(* PLC project Mx9_v_0_3_3.project, CODESYS CODESYS V3.5 SP5 Patch 5 *)
(* stored: creationDateTime 2017-10-23T23:21:49.9734832, modificationDateTime 2017-10-21T13:03:26.8127651 *)

TYPE component : STRUCT
  step : STRING;
  code : STRING;
  name : STRING;
  weight : STRING;
  roughWeight : STRING;
END_STRUCT;
END_TYPE

PROGRAM PLC_PRG
  VAR
    bStatInit : BOOL;
    bStatStandby : BOOL;
    bStatSettings : BOOL;
    bStatPause : BOOL;
    bStatLoad : BOOL;
    bLog : BOOL;
    bManualMode : BOOL;
    rTara : REAL;
    bTara : BOOL;
    rClean : REAL;
    precisionTimer : Standard.TON;
    sConsole : STRING := 'Console output';
    dfa : dfa;  (* classes *)
    switch : switch;
    list : list;
    logger : logger;
    recMan : RecipeManCommands;
    filter : filter;
  END_VAR

                    //a_read();
//b_tara();
rClean := filter.clean( rWeight );
blinkJob();
// test visu pumps to pump tubes link effect
FOR i := 1 TO 4 DO
	IF pumps[i] AND switch.isPumpRun() THEN pump_tubes[i] := TRUE; END_IF
END_FOR

CASE dfa.iStatementCode OF //набор состояний системы	
	0:// INIT
			blink ( TIMEHIGH := T#1S, TIMELOW := T#1S );
			bStatInit := TRUE;
			logger.init();
			recMan.WriteRecipe( namesGroup, namesFile );
			recMan.WriteRecipe( 'settings', filter_settngs_filename );
			dfa.exec('checked');
			
		IF dfa.bQuitStat THEN // EXIT
			bStatInit := FALSE;
		END_IF
		
	1:// STANDBY
		IF dfa.bEnterStat THEN
			 // ======== ENTER =========== //
			  //StatStandby := TRUE;
			//logger.writeStat( 'Enter standby mode');
			//IF logger.done THEN
				dfa.endEnter();
			//END_IF
			// ======== END ENTER ======== //
		END_IF
		
		//---------- BODY -----------//
		
		//------- END_BODY ----------//
		
		IF dfa.bQuitStat THEN 
		// ========== EXIT =========== //
			;
		// ======== END EXIT ======== //
		END_IF
		
	2:// SETTINGS
		IF dfa.bEnterStat THEN
			 // ======== ENTER =========== //
			 
			 
			dfa.endEnter();
			// ======== END ENTER ======== //
		END_IF
		
		//---------- BODY -----------//
		
		//------- END_BODY ----------//
		
		IF dfa.bQuitStat THEN 
		// ========== EXIT =========== //
		
		
		// ======== END EXIT ======== //
		END_IF

	3:// PROGRAMMING
		IF dfa.bEnterStat THEN
			 // ======== ENTER =========== //
			 
			 
			dfa.endEnter();
			// ======== END ENTER ======== //
		END_IF
		
		//---------- BODY -----------//
		
		//------- END_BODY ----------//
		
		IF dfa.bQuitStat THEN 
		// ========== EXIT =========== //
		
		
		// ======== END EXIT ======== //
		END_IF
		
	4:// CHOOSING
		IF dfa.bEnterStat THEN
			 // ======== ENTER =========== //
			dfa.endEnter();
			// ======== END ENTER ======== //
		END_IF
		
		//---------- BODY -----------//
		list.man_cmp_mode_job();
		//------- END_BODY ----------//
		
		IF dfa.bQuitStat THEN 
		// ========== EXIT =========== //
			IF bManualMode THEN
				list.man_counters_init();
			END_IF		
		// ======== END EXIT ======== //
		END_IF

	5:// ROUGH_LOADING
		IF dfa.bEnterStat THEN
			 // ======== ENTER =========== //
			IF bManualMode THEN 
				IF manWeightLimit = 0 THEN					
						dfa.exec('back'); 
					ELSE
						switch.on( componentNames[ i_man_count ], TRUE );
				END_IF
				
			END_IF
			 
			dfa.endEnter();
			// ======== END ENTER ======== //
		END_IF
		
		//---------- BODY -----------//
		IF bPause THEN dfa.exec('pause'); END_IF
		
		IF bManualMode THEN
			rWeight := rWeight + 0.01;
			list.man_mode_count();
			IF rWeight - rWeight_c_p >= ( manWeightLimit - manWeightPrecise ) THEN
				dfa.exec( 'done' );
			END_IF
		END_IF
		//------- END_BODY ----------//
		
		IF dfa.bQuitStat THEN 
		// ========== EXIT =========== //
		switch.allOff();
		
		// ======== END EXIT ======== //
		END_IF

	6:// PRECISE_LOADING
		IF dfa.bEnterStat THEN
			 // ======== ENTER =========== //
			dfa.endEnter();
			// ======== END ENTER ======== //
		END_IF
		
		//---------- BODY -----------//
		IF bPause THEN dfa.exec('pause'); END_IF
		
		IF bManualMode THEN
			precisionTimer( IN := TRUE, PT := T#5S );
			IF precisionTimer.Q THEN
				switch.on( componentNames[ i_man_count ], FALSE );
				rWeight := rWeight + 0.005;
				list.man_mode_count();
			END_IF
			IF rWeight - rWeight_c_p >= ( manWeightLimit ) THEN
				dfa.exec( 'listEnd' );
			END_IF
		END_IF
		//------- END_BODY ----------//
		
		IF dfa.bQuitStat THEN 
		// ========== EXIT =========== //
		precisionTimer( IN := FALSE );
		switch.allOff();
		
		// ======== END EXIT ======== //
		END_IF

	7:// DONE
		IF dfa.bEnterStat THEN
			 // ======== ENTER =========== //
			 
			dfa.endEnter();
			// ======== END ENTER ======== //
		END_IF		
		//---------- BODY -----------//
		
		//------- END_BODY ----------//
		
		IF dfa.bQuitStat THEN 
		// ========== EXIT =========== //
		
		
		// ======== END EXIT ======== //
		END_IF

	8:// PAUSE
		IF dfa.bEnterStat THEN
			 // ======== ENTER =========== //
				switch.allOff();
			 	logger.writeStat('Pause mode activated');
			 IF logger.done THEN
				dfa.endEnter();
			 END_IF
			// ======== END ENTER ======== //
		END_IF
		
		//---------- BODY -----------//
		IF NOT bPause THEN
			dfa.exec('back');			
			//switch.on( switch.sLastCode, switch.bLastRough );
		END_IF
		
		//------- END_BODY ----------//
		
		IF dfa.bQuitStat THEN 
		// ========== EXIT =========== //
		
		
		// ======== END EXIT ======== //
		END_IF

	ELSE	// состояние по-умолчанию
		
END_CASE
IF dfa.bQuitStat THEN // EXIT STATEMENT
	stats[dfa.iStatementCode] := FALSE;
	dfa.finishTransition();
	stats[dfa.iStatementCode] := TRUE;
END_IF
y_mach_table();
z_write();
                  

ACTION blinkJob:
                        IF switch.isPumpRun() THEN 
	blink( ENABLE := TRUE );		
	pumps[ switch.idxPump ] := blink.OUT ;
ELSE
	blink( ENABLE := FALSE );
END_IF
                      
END_ACTION

ACTION a_read:
                        rWeight := MV110_1TD.RdfF1 - rTara;
                      
END_ACTION

ACTION z_write:
                        iOutDiscrets := switch.iOut;
                      
END_ACTION

ACTION y_mach_table:
                        IF bManualMode THEN
	switch.matchTable();
END_IF;
                      
END_ACTION

ACTION b_tara:
                        IF bTara THEN
	rTara := MV110_1TD.RdfF1;
	bTara := FALSE;
END_IF
                      
END_ACTION
END_PROGRAM

FUNCTION_BLOCK dfa
  VAR_OUTPUT
    iStatementCode : INT;
    bEnterStat : BOOL;
    bQuitStat : BOOL;
  END_VAR
  VAR
    sCrntStatement : STRING := 'INIT';
    sPrevStatement : STRING;
    i : INT := 0;
    iFROM : INT := 0;
    iTRANSITION : INT := 1;
    iTO : INT := 2;
    arStatements : ARRAY[0..99] OF STRING := ['INIT', 'STANDBY', 'SETTINGS', 'PROGRAMMING', 'CHOOSING', 'ROUGH_LOADING', 'PRECISE_LOADING', 'DONE', 'PAUSE'];
    arTransitionTable : ARRAY[0..99, 0..2] OF STRING := ['INIT', 'checked', 'STANDBY', 'STANDBY', 'set', 'SETTINGS', 'STANDBY', 'start', 'CHOOSING', 'STANDBY', 'pause', 'PAUSE', 'SETTINGS', 'program', 'PROGRAMMING', 'SETTINGS', 'exit', 'STANDBY', 'PROGRAMMING', 'exit', 'STANDBY', 'PROGRAMMING', 'init', 'INIT', 'CHOOSING', 'exit', 'STANDBY', 'CHOOSING', 'load', 'ROUGH_LOADING', 'ROUGH_LOADING', 'pause', 'PAUSE', 'ROUGH_LOADING', 'done', 'PRECISE_LOADING', 'ROUGH_LOADING', 'listEnd', 'DONE', 'PRECISE_LOADING', 'next', 'ROUGH_LOADING', 'PRECISE_LOADING', 'pause', 'PAUSE', 'PRECISE_LOADING', 'listEnd', 'DONE', 'DONE', 'again', 'CHOOSING', 'DONE', 'exit', 'STANDBY', 'PAUSE', 'back', ''];
  END_VAR

                    
                  

{attribute 'object_name' := 'endEnter'}
METHOD endEnter
                          bEnterStat := FALSE;
                        
END_METHOD

{attribute 'object_name' := 'exec'}
METHOD exec
  VAR_INPUT
    sTransition : STRING;
  END_VAR
                          FOR i:= 0 TO 99 DO
	IF arTransitionTable[i, iFROM] = '' THEN
		RETURN;
	END_IF
	IF arTransitionTable[i, iFROM] = sCrntStatement AND arTransitionTable[i, iTRANSITION] = sTransition THEN
		
		sCrntStatement := SEL ( sTransition = 'back', arTransitionTable[i, iTO], sPrevStatement );
		
		sPrevStatement := arTransitionTable[i, iFROM];
		bQuitStat := TRUE;
		RETURN;
	END_IF
END_FOR
                        
END_METHOD

{attribute 'object_name' := 'finishTransition'}
METHOD finishTransition
                          FOR i:= 0 TO 99 DO
	IF arStatements[i] = '' THEN
		RETURN;		
	END_IF
	IF arStatements[i] = sCrntStatement THEN
		iStatementCode := i;
		bQuitStat := FALSE;
		bEnterStat := TRUE;
		RETURN;
	END_IF
END_FOR
                        
END_METHOD
END_FUNCTION_BLOCK

(* Набор переключателей *)
FUNCTION_BLOCK switch
  VAR_INPUT
    iIn : INT;
  END_VAR
  VAR_OUTPUT
    iOut : INT;
    idxPump : INT;
    sLastCode : STRING;
    bLastRough : BOOL;
  END_VAR
  VAR
    i : INT;
  END_VAR

                    
                  

(* выключает все 16 переключателей *)
{attribute 'object_name' := 'allOff'}
METHOD allOff
                          iOut := 0;
FOR i := 1 TO 11 DO
	IF i < 5 THEN
		pumps[ i ] := FALSE;
		pump_tubes[ i ] := FALSE;
	END_IF
	IF i < 10 THEN
		component_boxes[ i ] := FALSE;
	END_IF
	valves[ i ] := FALSE;
END_FOR
bPrecise := FALSE;
bRough := FALSE;
idxPump := 0;
                        
END_METHOD

(* устанавливает выключатели в ON *)
{attribute 'object_name' := 'on'}
METHOD on
  VAR_INPUT
    code : STRING;
    rough : BOOL;
  END_VAR
                          bRough := rough;
bPrecise := NOT rough;

sLastCode := code;
bLastRough := rough;

CASE getCodeIdx( code ) OF //набор переключателей в зависимости от кода
	1:	
			component_boxes[1] := TRUE;
			valves[1]	:= TRUE;
			valves[8]	:= TRUE;
			pump_tubes[1] := TRUE;
			idxPump := 1;			
	2:
			component_boxes[2] := TRUE;
			valves[2]	:= TRUE;
			valves[8]	:= TRUE;
			pump_tubes[1] := TRUE;
			idxPump := 1;			
	3:
			component_boxes[3] := TRUE;
			valves[3]	:= TRUE;
			valves[8]	:= TRUE;
			pump_tubes[1] := TRUE;
			idxPump := 1;
	4:
			component_boxes[4] := TRUE;
			valves[4]	:= TRUE;
			valves[8]	:= TRUE;
			pump_tubes[1] := TRUE;
			idxPump := 1;
	5:
			component_boxes[5] := TRUE;
			valves[5]	:= TRUE;
			valves[11]	:= TRUE;
			pump_tubes[2] := TRUE;
			idxPump := 2;
	6:
			component_boxes[6] := TRUE;
			valves[6]	:= TRUE;
			valves[11]	:= TRUE;
			pump_tubes[2] := TRUE;
			idxPump := 2;
	7:
			component_boxes[7] := TRUE;
			valves[7]	:= TRUE;
			valves[11]	:= TRUE;
			pump_tubes[2] := TRUE;
			idxPump := 2;
	8:
			component_boxes[8] := TRUE;
			valves[10]	:= TRUE;
			pump_tubes[3] := TRUE;
			idxPump := 3;
	9:
			component_boxes[9] := TRUE;
			valves[9]	:= TRUE;
			pump_tubes[4] := TRUE;
			idxPump := 4;
	;
	ELSE //	такого кода нет 
	//TODO - Error, example:
	error := 'ERROR: no such code of the ingredient. Program stopped.';
	showError := TRUE;
	allOff();
END_CASE
                        
END_METHOD

{attribute 'object_name' := 'getCodeIdx'}
METHOD getCodeIdx : INT
  VAR_INPUT
    code : STRING;
  END_VAR
                          FOR i := 1 TO 9 DO
	IF componentNames[i] = code THEN
		getCodeIdx := i;
		RETURN;
	END_IF
END_FOR
getCodeIdx :=  0;
                        
END_METHOD

{attribute 'object_name' := 'isPumpRun'}
METHOD isPumpRun : BOOL
                          isPumpRun := idxPump > 0 AND idxPump < 5;
                        
END_METHOD

{attribute 'object_name' := 'matchTable'}
METHOD matchTable
                          iOut.0:= component_boxes[1];
iOut.1:= component_boxes[2];
iOut.2 := component_boxes[3];
iOut.3 := component_boxes[4];
iOut.4 := component_boxes[5];
iOut.5 := component_boxes[6];
iOut.6 := component_boxes[7];
iOut.7 := component_boxes[8];
iOut.8 := component_boxes[9];

iOut.10 := bPrecise;
iOut.9 := bRough;
                        
END_METHOD
END_FUNCTION_BLOCK

FUNCTION_BLOCK list
  VAR_INPUT
    ptToSwitch : POINTER TO switch;
  END_VAR
  VAR
    bPrgDone : BOOL;  (* way:Way; *)
    bActive : BOOL;
    iPrgSteps : INT;
    iPrgIdx : INT;
    iLinePrgList : INT;
    iLine : INT;
    iTotalWeight : INT;
    iCleanIdx : INT;
    iCrntPoint : INT;
    iDirection : INT := 1;
    iArrLength : INT := 50;
    iPrgAmount : INT := 100;
  END_VAR

                    
                  

{attribute 'object_name' := 'getPrgIdx'}
METHOD getPrgIdx : INT
                          getPrgIdx := iLinePrgList;
                        
END_METHOD

{attribute 'object_name' := 'getLineFromPrgArr'}
METHOD getLineFromPrgArr : BOOL
  VAR_INPUT
    i : INT;
  END_VAR
                          (*currentIngredientName := arrayOfIngr[i].nameOfIngr;
currentWeight := STRING_TO_INT(arrayOfIngr[i].weightOfIngr);
//strCrntWay := arrayOfIngr[i].isDissolve;
way.setWay(arrayOfIngr[i].isDissolve);
ptToSwitch^.iWayIdx := way.getWayId();
currentTimeMixing := STRING_TO_TIME(arrayOfIngr[i].timeOfMixing);
message := arrayOfIngr[i].addMessage;*)
                        
END_METHOD

{attribute 'object_name' := 'stop'}
METHOD stop
                          bActive := FALSE;
iPrgIdx := 0;
                        
END_METHOD

{attribute 'object_name' := 'checkPrgArr'}
METHOD checkPrgArr : BOOL
                          (*currentProgramIdx:=0;
currentPrgSteps := 0;
iTotalWeight := 0;
IF LEN(arrayOfIngr[0].stepNum) = 0 THEN
		(* Поставить выброс ошибки в ответ на пустую или неправильную программу*)
		RETURN;		
END_IF
	
FOR iLine:= 0 TO 100 DO		
	IF 	LEN(arrayOfIngr[iLine].stepNum) > 0 THEN
		currentPrgSteps := currentPrgSteps + 1;
		iTotalWeight := iTotalWeight + STRING_TO_INT(arrayOfIngr[iLine].weightOfIngr);
		(* Поставить выброс ошибки если вес превышает максимально допустимый *)
	ELSE
		RETURN;	
	END_IF
END_FOR*)
                        
END_METHOD

{attribute 'object_name' := 'clearList'}
METHOD clearList : BOOL
                          (*FOR iCleanIdx:=0 TO iArrLength DO
	arrayOfIngr[iCleanIdx].stepNum:='';
	arrayOfIngr[iCleanIdx].nameOfIngr:='';
	arrayOfIngr[iCleanIdx].weightOfIngr:='';
	arrayOfIngr[iCleanIdx].isDissolve:='';
	arrayOfIngr[iCleanIdx].timeOfMixing:='';
	arrayOfIngr[iCleanIdx].addMessage:='';
END_FOR
 iCleanIdx:=0;
 iLine:=0;*)
                        
END_METHOD

{attribute 'object_name' := 'clearLine'}
METHOD clearLine : BOOL
                          (*IF iLine > 0 THEN
	iLine:=iLine - 1;
END_IF
arrayOfIngr[iLine].stepNum:='';
arrayOfIngr[iLine].nameOfIngr:='';
arrayOfIngr[iLine].weightOfIngr:='';
arrayOfIngr[iLine].isDissolve:='';
arrayOfIngr[iLine].timeOfMixing:='';
arrayOfIngr[iLine].addMessage:='';*)
                        
END_METHOD

{attribute 'object_name' := 'writeLine'}
METHOD writeLine : BOOL
                          (*
arrayOfIngr[iLine].stepNum := CONCAT('Step ', INT_TO_STRING(iLine+1));
arrayOfIngr[iLine].nameOfIngr := currentIngredientName;
arrayOfIngr[iLine].weightOfIngr := INT_TO_STRING(currentWeight);
arrayOfIngr[iLine].isDissolve := way.getWay();
currentTimeMixing := TimeInput(inputTime);
arrayOfIngr[iLine].timeOfMixing := TIME_TO_STRING(currentTimeMixing);
arrayOfIngr[iLine].addMessage := message;

iLine := iLine + 1;	
IF iLine > iArrLength THEN
	iLine := 0;
END_IF
*)
                        
END_METHOD

{attribute 'object_name' := 'keepGoing'}
METHOD keepGoing : BOOL
  VAR_INPUT
    iWeight : INT;
  END_VAR
                          keepGoing := FALSE;
                        
END_METHOD

{attribute 'object_name' := 'next'}
METHOD next
                          (*iPrgIdx := iPrgIdx + iDirection;
IF isLoad() AND iPrgIdx = iPrgSteps THEN
	turnBack();
END_IF
IF isUnload() AND iPrgIdx < 0 THEN
	stop();
	RETURN;
END_IF
getLineFromPrgArr(iPrgIdx);
iCrntPoint := iCrntPoint + (STRING_TO_INT(arrayOfIngr[iPrgIdx].weightOfIngr) * iDirection);*)
                        
END_METHOD

{attribute 'object_name' := 'start'}
METHOD start
                          (*bActive := TRUE;
iDirection := 1;
iPrgIdx := 0;
iPrgSteps := currentPrgSteps;
iCrntPoint := STRING_TO_INT(arrayOfIngr[iPrgIdx].weightOfIngr);
getLineFromPrgArr(iPrgIdx);*)
                        
END_METHOD

{attribute 'object_name' := 'man_cmp_mode_job'}
METHOD man_cmp_mode_job
                          FOR i := 1 TO 9 DO
	arr_cmpn_choosed[i] := FALSE;
END_FOR
arr_cmpn_choosed[iNames] := TRUE;
                        
END_METHOD

{attribute 'object_name' := 'clean_counters'}
METHOD clean_counters
                          FOR i := 1 TO 9 DO
	arr_cmpn_cnt[i] := 0;
	arr_cnt_crnt_points[i] := 0;
	rWeight_c_p := 0;
END_FOR
                        
END_METHOD

{attribute 'object_name' := 'man_mode_count'}
METHOD man_mode_count
                          arr_cmpn_cnt[ i_man_count ] := arr_cnt_crnt_points[ i_man_count ] + rWeight - rWeight_c_p;
                        
END_METHOD

{attribute 'object_name' := 'man_counters_init'}
METHOD man_counters_init
                          rWeight_c_p := rWeight;
arr_cnt_crnt_points[iNames] := arr_cmpn_cnt[iNames];
i_man_count := iNames;
                        
END_METHOD
END_FUNCTION_BLOCK

FUNCTION_BLOCK logger
  VAR_OUTPUT
    done : BOOL;
    date_Y_M_D : STRING;
  END_VAR
  VAR
    filename : FILE.CAA.FILENAME := LOG_FILE_PATH;
    message : STRING;
    xFileStdInit : BOOL := FALSE;
    uiFileStdState : UINT := 0;
    fOpen : FILE.Open;
    fWrite : FILE.Write;
    fRead : FILE.Read;
    fClose : FILE.Close;
    SetPos : FILE.SetPos;
    hFile : FILE.CAA.HANDLE;
    szFileSize : FILE.CAA.SIZE := 0;
  END_VAR

                    
                  

{attribute 'object_name' := 'exitLog'}
METHOD exitLog
                          xFileStdInit	:= FALSE;
uiFileStdState	:= 0;
                        
END_METHOD

{attribute 'object_name' := 'setPath'}
METHOD setPath
  VAR_INPUT
    path : STRING;
  END_VAR
                          filename := path;
                        
END_METHOD

{attribute 'object_name' := 'write'}
METHOD write : BOOL
  VAR_INPUT
    data : STRING;
  END_VAR
                          IF NOT xFileStdInit THEN
	done :=	FALSE;

	fOpen(xExecute:=FALSE);

	fClose(xExecute:=FALSE);

	fWrite(xExecute:=FALSE);

	fRead(xExecute:=FALSE);

	xFileStdInit:=TRUE;

	uiFileStdState:=0;

ELSE
	CASE uiFileStdState OF

		0: (* open file *)

         	fOpen.sFileName:= filename;
	
			fOpen.eFileMode:= FILE.MODE.MAPPD;

			fOpen.xExclusive:=TRUE;

			fOpen( xExecute:=TRUE );

				IF fOpen.xDone THEN

					hFile := fOpen.hFile;
					
					uiFileStdState := 2;

				END_IF

			   	IF fOpen.xError THEN (* error handling*)
					
					fOpen(xExecute:=FALSE);
					
					uiFileStdState := 1;

				  	error := 'error file opening, trying to create...' ;

			   	END_IF
				1:(* create file - if not exists *)

				   fOpen.eFileMode:= FILE.MODE.MWRITE;
				   
				   fOpen( xExecute:=TRUE );
				   
				   IF fOpen.xDone THEN
					   
						fOpen( xExecute := FALSE );
						
						uiFileStdState := 0;
						
						error := '';

					END_IF
					
					IF fOpen.xError THEN
						fOpen( xExecute := FALSE );
						
						uiFileStdState := 4;
	
						error := 'error file creating, log failed' ;

					END_IF

                2:(* write text in the file *)
					fWrite.hFile := hFile;
					message := Standard.CONCAT ( data, '$r' );
					message := Standard.CONCAT ( Standard.CONCAT ( now(), ' ' ) , message );
					fWrite.pBuffer:=ADR(message);
					szFileSize:= INT_TO_UINT( Standard.LEN( message ) );

					fWrite.szSize := szFileSize;
                               
				   	fWrite.udiTimeOut:=100000;                     (* 100ms Timeout *)

				   	fWrite( xExecute:=TRUE);

					   IF fWrite.xDone THEN
						   
						   SetPos( hFile := hFile, udiPos := 2);
	
						   uiFileStdState:=3;

					   END_IF

					   IF fWrite.xError THEN

									   (* error handling*)

									   ;

					   END_IF

                
                3:             (* close file  *)

					   fClose.hFile:= hFile;

					   fClose( xExecute:=TRUE);

					   IF fClose.xDone THEN

									   uiFileStdState:=4;

					   END_IF

					   IF fClose.xError THEN

									   (* error handling*)

									   ;

					   END_IF

				4:   (* end of log *)
						exitLog();
						done  := TRUE;
                END_CASE


END_IF
                        
END_METHOD

{attribute 'object_name' := 'now'}
METHOD now : STRING
  VAR
    Date_and_time_in_seconds : UDINT;  (* now timestamp *)
    Local_date_time_seconds : UDINT;
    Date_and_Time_result : UDINT;
    Local_date_time_from_secs : SYSTIMEDATE;
    Date_and_time_format : DT;
    Date_and_time_string : STRING;
  END_VAR
                          // Get time in seconds since 1970 :
Date_and_time_in_seconds := SysTimeRtcGet(Date_and_Time_result);
IF Date_and_Time_result <> 0 THEN
RETURN;
END_IF

// Convert UTC seconds to local time seconds, regarding Timezone and Summer time :
Date_and_Time_result := SysTimeRtcConvertUtcToLocal(Date_and_time_in_seconds, Local_date_time_seconds);
IF Date_and_Time_result <> 0 THEN
RETURN;
END_IF

// Convert the UTC seconds to a DATE_AND_TIME variable dt#yyyy-mm-dd-hh:mm:ss :
Date_and_time_format := UDINT_TO_DT(Local_date_time_seconds);

// Convert DATE_AND_TIME to a String :
Date_and_time_string := DT_TO_STRING(Date_and_time_format);

date_Y_M_D := Standard.MID( Date_and_time_string, 10, 4 );

now := REPLACE ( Date_and_time_string, '', 3, 1 );
                        
END_METHOD

{attribute 'object_name' := 'writeStat'}
METHOD writeStat
  VAR_INPUT
    data : STRING;
  END_VAR
                          setPath( STAT_FILE_PATH );
write( data );
setPath( LOG_FILE_PATH );
                        
END_METHOD

{attribute 'object_name' := 'init'}
METHOD init
                          now();
LOG_FILE_PATH := Standard.CONCAT ( Standard.CONCAT( LOG_FILE_PATH, date_Y_M_D ), '.txt');
STAT_FILE_PATH := Standard.CONCAT ( Standard.CONCAT( STAT_FILE_PATH, date_Y_M_D ), '.txt');
                        
END_METHOD
END_FUNCTION_BLOCK

FUNCTION_BLOCK filter
  VAR_INPUT
    rIn : REAL;
  END_VAR
  VAR_OUTPUT
    rOut : REAL;
  END_VAR
  VAR
    arr : ARRAY[0..99] OF REAL;
    i : INT;
    arMax : REAL;
    arMin : REAL;
    rFixed : REAL;
  END_VAR

                    
                  

{attribute 'object_name' := 'array_push'}
METHOD array_push
  VAR_INPUT
    rInValue : REAL;
  END_VAR
  VAR
    i : INT;
  END_VAR
                          arMax := arr[filter_arr_length]; arMin := arr[filter_arr_length];
FOR i := filter_arr_length TO 0 BY -1 DO
	arMax := MAX ( arr[i], arMax );
	arMin := MIN ( arr[i], arMin );
	arr[i] := SEL ( i = 0, arr[i - 1], rInValue );
END_FOR
                        
END_METHOD

{attribute 'object_name' := 'isStable'}
METHOD isStable : BOOL
  VAR_INPUT
    rInput : REAL;
  END_VAR
                          isStable := 
		arMax >= arMin
	AND ABS ( arMax - arMin ) <= filter_channel_width  
	AND	ABS ( rInput - rFixed ) <= flter_stability_koef
;
                        
END_METHOD

{attribute 'object_name' := 'clean'}
METHOD clean : REAL
  VAR_INPUT
    rRaw : REAL;
  END_VAR
                          IF isStable( rRaw ) THEN
	filter_stable_int := SEL ( filter_stable_int >= filter_arr_length * 2, filter_stable_int + 1, filter_stable_int ) ;
	clean := rFixed;
	IF filter_stable_int >= filter_arr_length * 2 THEN
		RETURN;
	END_IF
ELSE
	filter_stable_int := 0;
END_IF
array_push( rRaw );
rFixed := count();
clean := rRaw;
                        
END_METHOD

{attribute 'object_name' := 'count'}
METHOD count : REAL
  VAR
    i : INT;
    sum : REAL;
  END_VAR
                          FOR i := 0 TO filter_arr_length DO
	sum := sum + arr[i];
END_FOR
count := sum / ABS ( filter_arr_length + 1 );
                        
END_METHOD
END_FUNCTION_BLOCK

CONFIGURATION Device
  RESOURCE Application ON PLC
    VAR_GLOBAL  (* config - путь для сохранения файлов в контроллере СПК 207 = /mnt/ufs/media/mmcblk0p1/ or /mnt/ufs/media/sda1/ путь для сохранения логов в контроллере СПК 207 = '/mnt/ufs/media/mmcblk0p1/log/' путь для сохранения статистики в контроллере СПК 207 = '/mnt/ufs/media/mmcblk0p1/stat/' путь для сохранения файлов в компьютере = C:\tmp\testRecipe путь для сохранения логов в компьютере = 'C:\tmp\log\' путь для сохранения статистики в компьютере = 'C:\tmp\stat\' *)
      crComponent : component;  (* constants, global vars *)
      rWeight : REAL;
      rWeight_c_p : REAL;
      componentNames : ARRAY[1..9] OF STRING := ['alfa', 'bravo', 'charlie', 'delta', 'echo', 'foxtrot', 'golf', 'hotel', 'india'];
      iNames : UINT := 1;
      components : ARRAY[1..50] OF component;
      com_idx : INT := 1;
      i : UINT;  (* index for loop iterations *)
      arr_cmpn_cnt : ARRAY[0..9] OF REAL;  (* MANUAL MODE VARS *)
      i_man_count : UINT;
      arr_cnt_crnt_points : ARRAY[0..9] OF REAL;
      arr_cmpn_choosed : ARRAY[0..9] OF BOOL;
      i_cmp_cnt : INT;
      manWeightLimit : INT;
      manWeightPrecise : INT;
      filter_settngs_filename : STRING := 'filter';  (* SETTINGS *)
      filter_arr_length : INT := 99;
      filter_channel_width : REAL := 10;
      filter_stable_int : INT := 100;
      flter_stability_koef : REAL := 2;  (* distance between input signal and fixed value inside channel array *)
      iOutDiscrets : INT;  (* OUTER DATA *)
      MAX_WEIGHT : INT := 1000;  (* SYSTEM LIMITS *)
      MIN_WEIGHT : INT := 0;
      recipeName : STRING := 'Receipt';  (* WORK WITH FILESYSTEM *)
      namesGroup : STRING := 'names';
      namesFile : STRING := 'component';
      LOG_FILE_PATH : STRING := 'C:\tmp\log\';  (* logger files path, upated each progam start due to curent date *)
      STAT_FILE_PATH : STRING := 'C:\tmp\stat\';
      info : STRING;  (* handle errors, exceptions, inform message *)
      warning : STRING;
      error : STRING;
      showError : BOOL;
      bErorTextColor : BOOL;
      bPause : BOOL;  (* buttons *)
      bRoughBtn : BOOL := FALSE;
      bPreciseBtn : BOOL := FALSE;
      stats : ARRAY[0..9] OF BOOL;  (* statements indicator *)
      blink : BLINK;  (* single blink for pump indicate *)
      pumps : ARRAY[1..4] OF BOOL;  (* switches for screen activity *)
      pump_tubes : ARRAY[1..4] OF BOOL;
      valves : ARRAY[1..11] OF BOOL;
      component_boxes : ARRAY[1..9] OF BOOL;
      bPrecise : BOOL := FALSE;
      bRough : BOOL := FALSE;
    END_VAR
    TASK MainTask(INTERVAL := T#10ms, PRIORITY := 1);
    TASK VISU_TASK(INTERVAL := T#100ms, PRIORITY := 10);
    PROGRAM PLC_PRG WITH MainTask : PLC_PRG;
    PROGRAM VisuElems.Visu_Prg WITH VISU_TASK : VisuElems.Visu_Prg;
  END_RESOURCE
END_CONFIGURATION

CONFIGURATION COM_3
END_CONFIGURATION

CONFIGURATION Modbus_Master_COM_Port
END_CONFIGURATION

CONFIGURATION MV110_1TD
END_CONFIGURATION

CONFIGURATION Out_MU110_16R
END_CONFIGURATION
